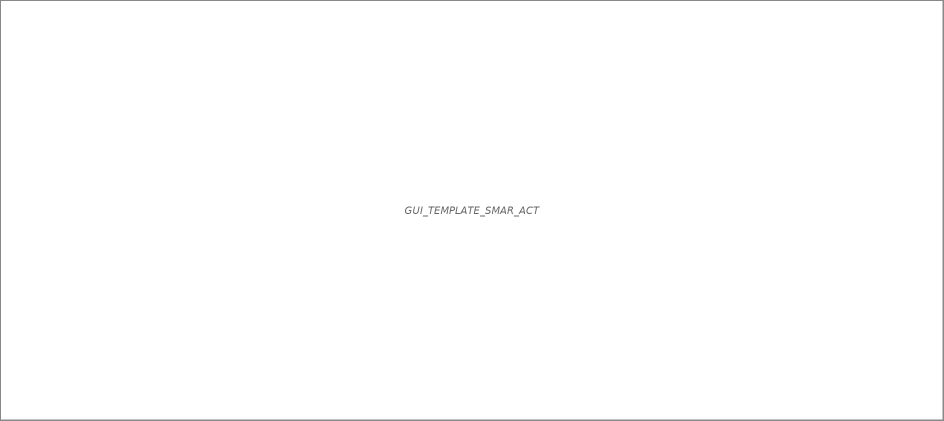
VISUALIZATION GUI_SmarAct_PDS  // 944x421
    Frame (0,0 944x421)
        shows GUI_TEMPLATE_SMAR_ACT(m_Instance := MAIN.SmarAct_PDS)
END_VISUALIZATION

(* stored: Version 1.1.0.1, ProductVersion 3.1.4024.10
   Visu GUI_SmarAct_PDS: Id {47054995-4266-4601-9076-76722ab40b8b} *)
